// RUN THE ALARM CHECK

FUNCTION RunAlarmCheck

VAR
	// Threashold value (both tests just happen to use the same value)
	thresh : REAL := 90;
	
	// FILL is alarm?
	h : BOOL := High.full_percent > thresh;
	
	// TEMP is alarm?
	t : BOOL := Temp.now > thresh;
	
END_VAR

status.alarm := h OR t;

END_FUNCTION

(* stored: Version 1.1.0.1, ProductVersion 3.1.4024.12
   POU RunAlarmCheck: Id {ce410715-b7c9-458a-8e35-072a529c7159}, SpecialFunc None *)
